{attribute 'linkalways'} 
{attribute 'no_explicit_call' := 'This FB is a CLASS and must be accessed using methods or properties'}
{attribute 'enable_dynamic_creation'}
FUNCTION_BLOCK SafeMemCopyOperation EXTENDS Disposable IMPLEMENTS I_DatatypeOperation
VAR
	source : I_Datatype;
	destination : I_Datatype;
END_VAR

METHOD Execute
VAR
END_VAR
destination.TryCopyFrom(source);
END_METHOD

METHOD FB_init : BOOL
VAR_INPUT
	bInitRetains : BOOL; // if TRUE, the retain variables are initialized (warm start / cold start)
	bInCopyCode : BOOL;  // if TRUE, the instance afterwards gets moved into the copy code (online change)
	Source : I_Datatype;
	Destination : I_Datatype;
END_VAR
THIS^.source := Source;
This^.destination := Destination;
END_METHOD

END_FUNCTION_BLOCK

(* stored: Version 1.1.0.1, ProductVersion 3.1.4024.12
   POU SafeMemCopyOperation: Id {9743687e-ddf5-4eb0-a0d2-01d50dd64dd7}, SpecialFunc None
   Folder Constructor: Id {878c6cbf-ae12-4735-92d9-bb7624ba633b}
   Method Execute: Id {02cf43c8-98d3-4ef5-a835-ab4c33d736fa}
   Method FB_init: Id {ea101a8f-0b98-43b2-80a1-0ec3450bd113} *)
